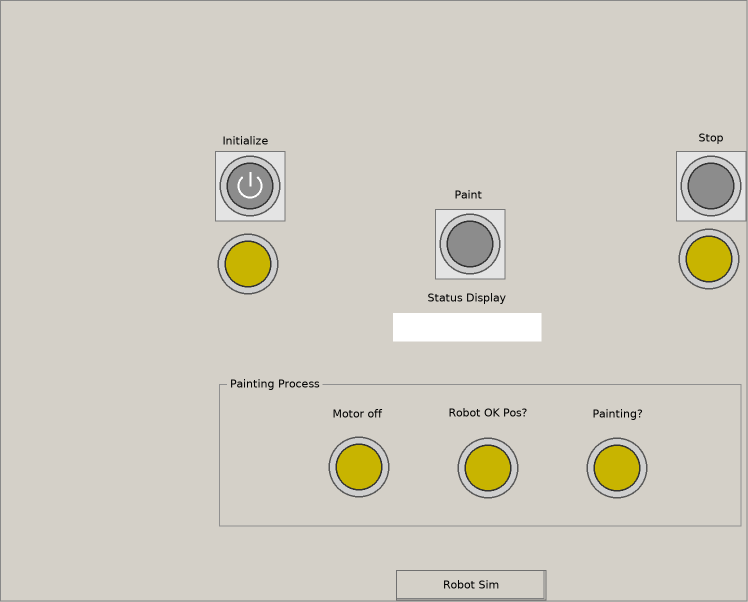
VISUALIZATION PaintVisualization  // 748x602
    GroupBox (219,376 522x150), "Painting Process"
        Label (92,18 93x40), "Motor off"
        Label (195,17 148x40), "Robot OK Pos?"
        Lamp1 (234,57 70x70), variable: Variables.bIsRobotInPos, style: Lamp-Lamp1-Yellow
        Lamp1 (105,56 70x70), style: Lamp-Lamp1-Yellow
    Lamp1 (213,229 70x70), variable: Variables.bSwitchON, style: Lamp-Lamp1-Yellow
    PushSwitch (676,151 70x70), variable: Variables.bStopOperations, behaviour: TOGGLE, style: Switch-PushSwitch-Gray
    Label (213,126 65x30), "Initialize"
    Label (685,123 52x30), "Stop"
    Lamp1 (582,433 70x70), style: Lamp-Lamp1-Yellow
    Label (541,399 154x30), "Painting?"
    PushSwitchLed (435,209 70x70), variable: Variables.bPaint, behaviour: TOGGLE, style: Switch-PushSwitchLed-Gray
    Label (436,180 65x30), "Paint"
    Textfield (392,312 150x30), text variable: Display.status_display
    Label (392,283 150x30), "Status Display"
    Lamp1 (674,224 70x70), variable: Variables.bStopOperations, style: Lamp-Lamp1-Yellow
    PowerSwitch (215,151 70x70), variable: Variables.bSwitchON, behaviour: TOGGLE, style: Switch-PowerSwitch-Gray
    Button (396,570 150x30), "Robot Sim"
        tap Variables.bIsRobotInPos
END_VISUALIZATION

(* stored: Version 1.1.0.1, ProductVersion 3.1.4020.6
   Visu PaintVisualization: Id {8d10fefd-042c-4d01-8a68-43092d8866c3} *)
